// TIA Portal V20 export
DATA_BLOCK "GLOBAL_INFO_FB_IDB"   // DB30231
AUTHOR : Tesla
FAMILY : Base
VERSION : 1.0
// stored: AutoNumber false, InstanceOfName GLOBAL_INFO_FB, InstanceOfType FB
"GLOBAL_INFO_FB"
   // VAR_INPUT
   //    NO_OPERATION_MODE { ExternalAccessible := 'False'; ExternalVisible := 'False'; ExternalWritable := 'False'} : Int;
   //    NO_HMI_PANEL { ExternalAccessible := 'False'; ExternalVisible := 'False'; ExternalWritable := 'False'} : Int;
   //    CLOCK_MEMORY { ExternalAccessible := 'False'; ExternalVisible := 'False'; ExternalWritable := 'False'} : Byte;
   //    SYSTEM_MEMORY { ExternalAccessible := 'False'; ExternalVisible := 'False'; ExternalWritable := 'False'} : Byte;
   //    RTG1SYSINFO { ExternalAccessible := 'False'; ExternalVisible := 'False'; ExternalWritable := 'False'} : F_SYSINFO;
   //    LADDR : HW_IO;
   // END_VAR
   // VAR_OUTPUT
   //    "ALWAYS=TRUE" { ExternalAccessible := 'False'; ExternalVisible := 'False'; ExternalWritable := 'False'} : Bool;
   //    "ALWAYS=FALSE" { ExternalAccessible := 'False'; ExternalVisible := 'False'; ExternalWritable := 'False'} : Bool;
   //    FIRST_CYCLE { ExternalAccessible := 'False'; ExternalVisible := 'False'; ExternalWritable := 'False'} : Bool;
   // END_VAR
   // VAR_IN_OUT
   //    INIT_HMI_OPMODE : "INIT_HMI_OPMODE_UDT";
   // END_VAR
   // VAR
   //    HMI_GLOBAL { S7_SetPoint := 'True'} : "GLOBAL_STRUCT_UDT";
   //    HMI_ClockMemory : Byte;
   // END_VAR
BEGIN
END_DATA_BLOCK
